{attribute 'GeneratedUsingTerminal: KL9940-0050'}
{attribute addProperty BoxType "KL9940-0050"}
{attribute addProperty Id "Key_1AT %I*BOOL0Key_2AT %I*BOOL0Key_3AT %I*BOOL0Key_4AT %I*BOOL0Key_5AT %I*BOOL0Key_6AT %I*BOOL0Key_7AT %I*BOOL0Key_8AT %I*BOOL0Key_9AT %I*BOOL0Key_10AT %I*BOOL0Key_11AT %I*BOOL0Key_12AT %I*BOOL0Key_13AT %I*BOOL0Key_14AT %I*BOOL0Key_15AT %I*BOOL0Key_16AT %I*BOOL0Key_17AT %I*BOOL0Key_18AT %I*BOOL0Key_19AT %I*BOOL0Key_20AT %I*BOOL0Key_21AT %I*BOOL0Key_22AT %I*BOOL0Key_23AT %I*BOOL0Key_24AT %I*BOOL0Key_25AT %I*BOOL0Key_26AT %I*BOOL0Key_27AT %I*BOOL0Key_28AT %I*BOOL0Key_29AT %I*BOOL0Key_30AT %I*BOOL0Key_31AT %I*BOOL0Key_32AT %I*BOOL0Key_33AT %I*BOOL0Key_34AT %I*BOOL0Key_35AT %I*BOOL0Key_36AT %I*BOOL0Key_37AT %I*BOOL0Key_38AT %I*BOOL0Key_39AT %I*BOOL0Key_40AT %I*BOOL0"}
{attribute addProperty CRC "2504797933"}
{attribute addProperty Size "0"}
TYPE Channel_954C2EED :
STRUCT
	{attribute addProperty Name "Key_1"}
	Key_1 AT %I* : BOOL;
	{attribute addProperty Name "Key_2"}
	Key_2 AT %I* : BOOL;
	{attribute addProperty Name "Key_3"}
	Key_3 AT %I* : BOOL;
	{attribute addProperty Name "Key_4"}
	Key_4 AT %I* : BOOL;
	{attribute addProperty Name "Key_5"}
	Key_5 AT %I* : BOOL;
	{attribute addProperty Name "Key_6"}
	Key_6 AT %I* : BOOL;
	{attribute addProperty Name "Key_7"}
	Key_7 AT %I* : BOOL;
	{attribute addProperty Name "Key_8"}
	Key_8 AT %I* : BOOL;
	{attribute addProperty Name "Key_9"}
	Key_9 AT %I* : BOOL;
	{attribute addProperty Name "Key_10"}
	Key_10 AT %I* : BOOL;
	{attribute addProperty Name "Key_11"}
	Key_11 AT %I* : BOOL;
	{attribute addProperty Name "Key_12"}
	Key_12 AT %I* : BOOL;
	{attribute addProperty Name "Key_13"}
	Key_13 AT %I* : BOOL;
	{attribute addProperty Name "Key_14"}
	Key_14 AT %I* : BOOL;
	{attribute addProperty Name "Key_15"}
	Key_15 AT %I* : BOOL;
	{attribute addProperty Name "Key_16"}
	Key_16 AT %I* : BOOL;
	{attribute addProperty Name "Key_17"}
	Key_17 AT %I* : BOOL;
	{attribute addProperty Name "Key_18"}
	Key_18 AT %I* : BOOL;
	{attribute addProperty Name "Key_19"}
	Key_19 AT %I* : BOOL;
	{attribute addProperty Name "Key_20"}
	Key_20 AT %I* : BOOL;
	{attribute addProperty Name "Key_21"}
	Key_21 AT %I* : BOOL;
	{attribute addProperty Name "Key_22"}
	Key_22 AT %I* : BOOL;
	{attribute addProperty Name "Key_23"}
	Key_23 AT %I* : BOOL;
	{attribute addProperty Name "Key_24"}
	Key_24 AT %I* : BOOL;
	{attribute addProperty Name "Key_25"}
	Key_25 AT %I* : BOOL;
	{attribute addProperty Name "Key_26"}
	Key_26 AT %I* : BOOL;
	{attribute addProperty Name "Key_27"}
	Key_27 AT %I* : BOOL;
	{attribute addProperty Name "Key_28"}
	Key_28 AT %I* : BOOL;
	{attribute addProperty Name "Key_29"}
	Key_29 AT %I* : BOOL;
	{attribute addProperty Name "Key_30"}
	Key_30 AT %I* : BOOL;
	{attribute addProperty Name "Key_31"}
	Key_31 AT %I* : BOOL;
	{attribute addProperty Name "Key_32"}
	Key_32 AT %I* : BOOL;
	{attribute addProperty Name "Key_33"}
	Key_33 AT %I* : BOOL;
	{attribute addProperty Name "Key_34"}
	Key_34 AT %I* : BOOL;
	{attribute addProperty Name "Key_35"}
	Key_35 AT %I* : BOOL;
	{attribute addProperty Name "Key_36"}
	Key_36 AT %I* : BOOL;
	{attribute addProperty Name "Key_37"}
	Key_37 AT %I* : BOOL;
	{attribute addProperty Name "Key_38"}
	Key_38 AT %I* : BOOL;
	{attribute addProperty Name "Key_39"}
	Key_39 AT %I* : BOOL;
	{attribute addProperty Name "Key_40"}
	Key_40 AT %I* : BOOL;
END_STRUCT
END_TYPE

(* stored: Version 1.2.0.0, ProductVersion 3.1.4024.9
   DUT Channel_954C2EED: Id {ab66613b-34be-44fc-a3c2-cc3155340830} *)
